(* PLC project Unnamed, Unknown Unnamed 1 *)
(* stored: creationDateTime 2023-03-10T10:37:17, modificationDateTime 2023-03-15T15:56:42 *)

(* 978-3-658-16137-8, Aufgabe 2.42 *)
FUNCTION_BLOCK Ventilation_Control_System
  VAR_INPUT
    IN1 : BOOL;
    IN2 : BOOL;
    IN3 : BOOL;
    IN4 : BOOL;
  END_VAR
  VAR_OUTPUT
    OUT1 : BOOL;
    OUT2 : BOOL;
    OUT3 : BOOL;
  END_VAR

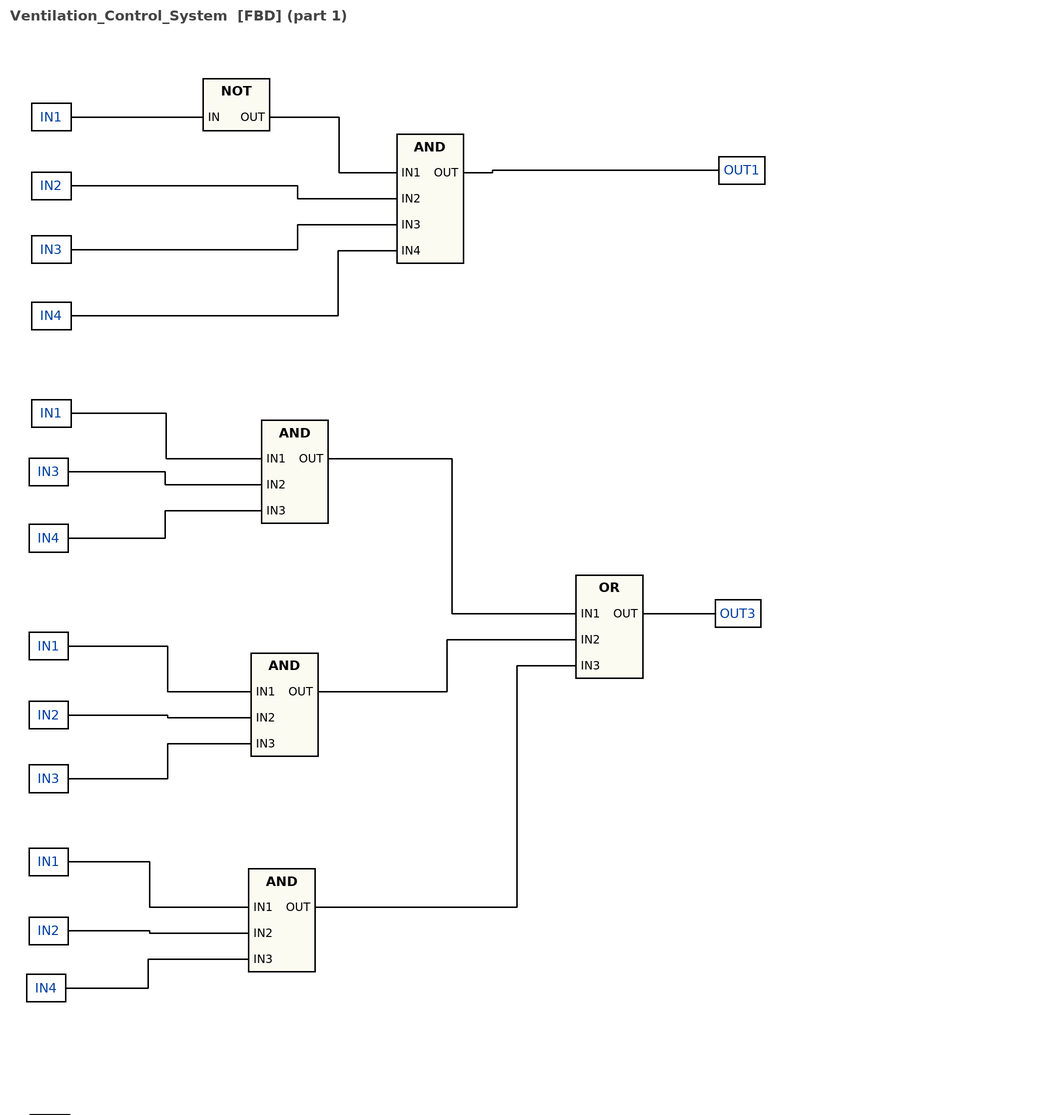
(* FBD diagram, written out as Structured Text *)
OUT1 := NOT IN1 AND IN2 AND IN3 AND IN4;
OUT3 := IN1 AND IN3 AND IN4 OR IN1 AND IN2 AND IN3 OR IN1 AND IN2 AND IN4;
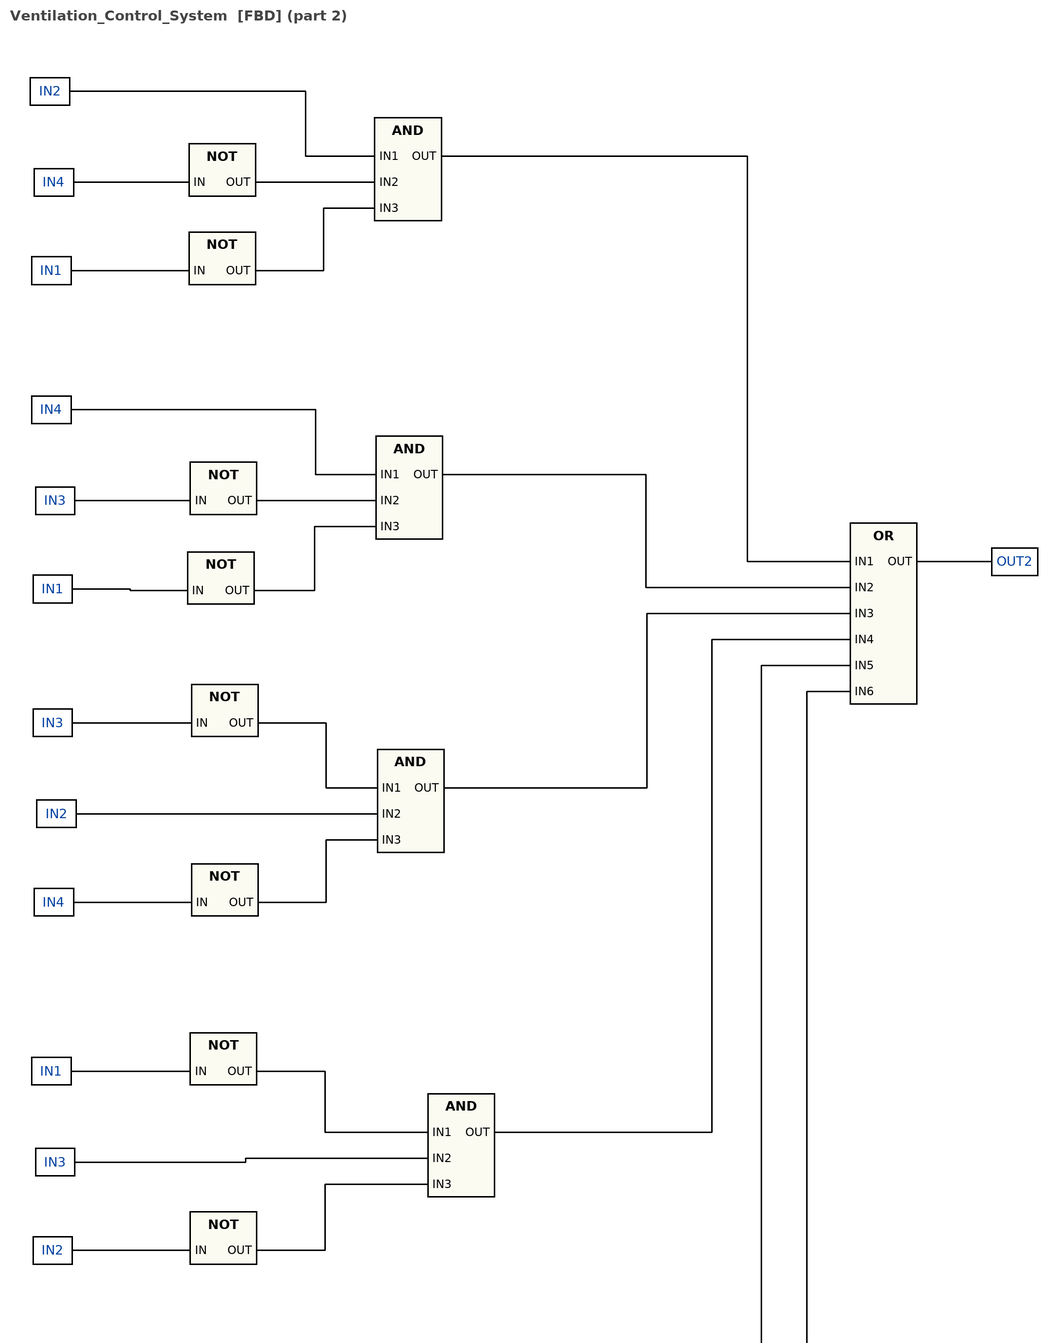
OUT2 := IN2 AND NOT IN4 AND NOT IN1 OR IN4 AND NOT IN3 AND NOT IN1 OR NOT IN3 AND IN2 AND NOT IN4 OR NOT IN1 AND IN3 AND NOT IN2 OR NOT IN4 AND IN1 AND NOT IN2 OR NOT IN3 AND IN1 AND NOT IN2;
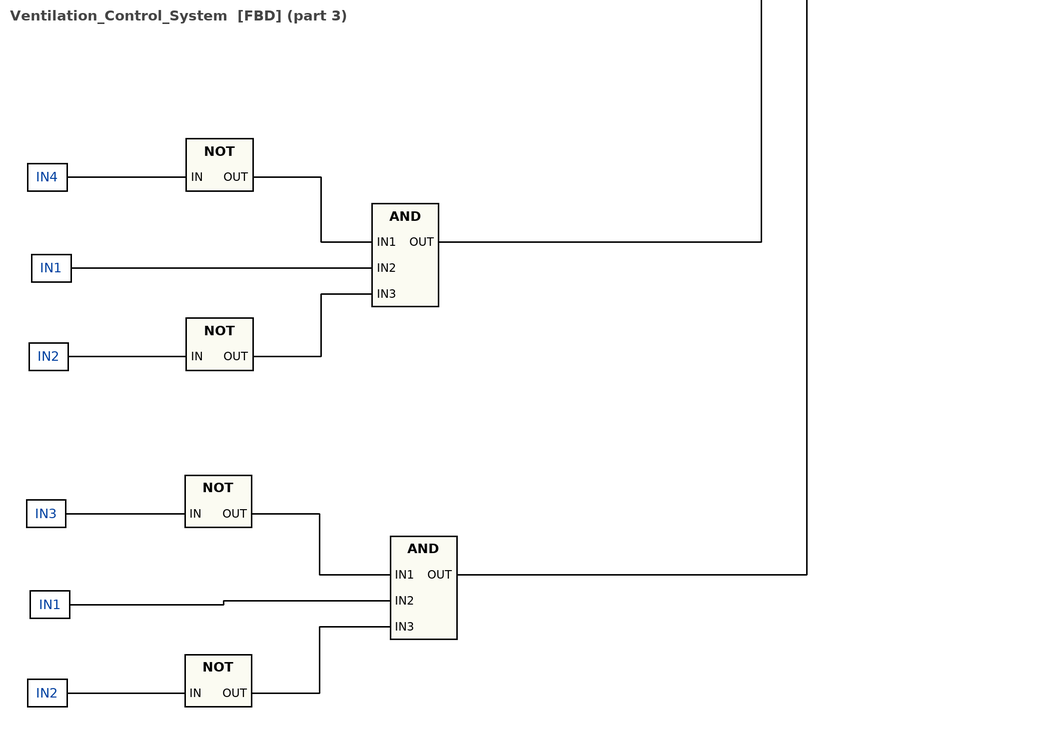
END_FUNCTION_BLOCK

CONFIGURATION config
  RESOURCE resource1 ON PLC
  END_RESOURCE
END_CONFIGURATION
